(*
Nazwa:			FB_OEECycleTimes
Opis:			czasy cyklów
Wersja:			v0.1
Data:			2021-11-09
Autor:			DP
Urzadzenia:		
Konfiguracja:	
Info: 
- dodano opcje przesuwu liniowego
*)
FUNCTION_BLOCK FB_OEECycleTimes
VAR_INPUT
	bEnable: BOOL;				//Zezwolenie na pracę
	bReset:BOOL;				//Stop awaryjny nieaktywny
	tStation1CT:TIME;			//Czas cyklu stacji nr 1
	bStation1En:BOOL;			//Zezwolenie pracy stacji nr 1
	sStation1Name:STRING;		//Nazwa stacji nr 1
	tStation2CT:TIME;			//Czas cyklu stacji nr 2
	bStation2En:BOOL;			//Zezwolenie pracy stacji nr 2
	sStation2Name:STRING;		//Nazwa stacji nr 2
	tStation3CT:TIME;			//Czas cyklu stacji nr 3
	bStation3En:BOOL;			//Zezwolenie pracy stacji nr 3
	sStation3Name:STRING;		//Nazwa stacji nr 3
	tStation4CT:TIME;			//Czas cyklu stacji nr 4
	bStation4En:BOOL;			//Zezwolenie pracy stacji nr 4
	sStation4Name:STRING;		//Nazwa stacji nr 4
	tStation5CT:TIME;			//Czas cyklu stacji nr 5
	bStation5En:BOOL;			//Zezwolenie pracy stacji nr 5
	sStation5Name:STRING;		//Nazwa stacji nr 5
	tStation6CT:TIME;			//Czas cyklu stacji nr 6
	bStation6En:BOOL;			//Zezwolenie pracy stacji nr 6
	sStation6Name:STRING;		//Nazwa stacji nr 6
	tStation7CT:TIME;			//Czas cyklu stacji nr 7
	bStation7En:BOOL;			//Zezwolenie pracy stacji nr 7
	sStation7Name:STRING;		//Nazwa stacji nr 7
	tStation8CT:TIME;			//Czas cyklu stacji nr 8
	bStation8En:BOOL;			//Zezwolenie pracy stacji nr 8
	sStation8Name:STRING;		//Nazwa stacji nr 8
	tStation9CT:TIME;			//Czas cyklu stacji nr 9
	bStation9En:BOOL;			//Zezwolenie pracy stacji nr 9
	sStation9Name:STRING;		//Nazwa stacji nr 9
	tStation10CT:TIME;			//Czas cyklu stacji nr 10
	bStation10En:BOOL;			//Zezwolenie pracy stacji nr 10
	sStation10Name:STRING;		//Nazwa stacji nr 10
	tStation11CT:TIME;			//Czas cyklu stacji nr 11
	bStation11En:BOOL;			//Zezwolenie pracy stacji nr 11
	sStation11Name:STRING;		//Nazwa stacji nr 11
	tStation12CT:TIME;			//Czas cyklu stacji nr 12
	bStation12En:BOOL;			//Zezwolenie pracy stacji nr 12
	sStation12Name:STRING;		//Nazwa stacji nr 12
	tStation13CT:TIME;			//Czas cyklu stacji nr 13
	bStation13En:BOOL;			//Zezwolenie pracy stacji nr 13
	sStation13Name:STRING;		//Nazwa stacji nr 13
	tStation14CT:TIME;			//Czas cyklu stacji nr 14
	bStation14En:BOOL;			//Zezwolenie pracy stacji nr 14
	sStation14Name:STRING;		//Nazwa stacji nr 14
	tStation15CT:TIME;			//Czas cyklu stacji nr 15
	bStation15En:BOOL;			//Zezwolenie pracy stacji nr 15	
	sStation15Name:STRING;		//Nazwa stacji nr 15
	tStation16CT:TIME;			//Czas cyklu stacji nr 16
	bStation16En:BOOL;			//Zezwolenie pracy stacji nr 16	
	sStation16Name:STRING;		//Nazwa stacji nr 16
	tStation17CT:TIME;			//Czas cyklu stacji nr 17
	bStation17En:BOOL;			//Zezwolenie pracy stacji nr 17	
	sStation17Name:STRING;		//Nazwa stacji nr 17
	tStation18CT:TIME;			//Czas cyklu stacji nr 18
	bStation18En:BOOL;			//Zezwolenie pracy stacji nr 18	
	sStation18Name:STRING;		//Nazwa stacji nr 18
	tStation19CT:TIME;			//Czas cyklu stacji nr 19
	bStation19En:BOOL;			//Zezwolenie pracy stacji nr 19	
	sStation19Name:STRING;		//Nazwa stacji nr 19
	tStation20CT:TIME;			//Czas cyklu stacji nr 20
	bStation20En:BOOL;			//Zezwolenie pracy stacji nr 20	
	sStation20Name:STRING;		//Nazwa stacji nr 20
	tStation21CT:TIME;			//Czas cyklu stacji nr 21
	bStation21En:BOOL;			//Zezwolenie pracy stacji nr 21	
	sStation21Name:STRING;		//Nazwa stacji nr 21	
	tStation22CT:TIME;			//Czas cyklu stacji nr 22
	bStation22En:BOOL;			//Zezwolenie pracy stacji nr 22	
	sStation22Name:STRING;		//Nazwa stacji nr 22	
	tStation23CT:TIME;			//Czas cyklu stacji nr 23
	bStation23En:BOOL;			//Zezwolenie pracy stacji nr 23	
	sStation23Name:STRING;		//Nazwa stacji nr 23	
	tStation24CT:TIME;			//Czas cyklu stacji nr 24
	bStation24En:BOOL;			//Zezwolenie pracy stacji nr 24	
	sStation24Name:STRING;		//Nazwa stacji nr 24	
	tStation25CT:TIME;			//Czas cyklu stacji nr 25
	bStation25En:BOOL;			//Zezwolenie pracy stacji nr 25	
	sStation25Name:STRING;		//Nazwa stacji nr 25	
	tStation26CT:TIME;			//Czas cyklu stacji nr 26
	bStation26En:BOOL;			//Zezwolenie pracy stacji nr 26	
	sStation26Name:STRING;		//Nazwa stacji nr 26	
	tStation27CT:TIME;			//Czas cyklu stacji nr 27
	bStation27En:BOOL;			//Zezwolenie pracy stacji nr 27	
	sStation27Name:STRING;		//Nazwa stacji nr 27	
	tStation28CT:TIME;			//Czas cyklu stacji nr 28
	bStation28En:BOOL;			//Zezwolenie pracy stacji nr 28	
	sStation28Name:STRING;		//Nazwa stacji nr 28	
	tStation29CT:TIME;			//Czas cyklu stacji nr 29
	bStation29En:BOOL;			//Zezwolenie pracy stacji nr 29	
	sStation29Name:STRING;		//Nazwa stacji nr 29	
	tStation30CT:TIME;			//Czas cyklu stacji nr 30
	bStation30En:BOOL;			//Zezwolenie pracy stacji nr 30	
	sStation30Name:STRING;		//Nazwa stacji nr 30	
	tStation31CT:TIME;			//Czas cyklu stacji nr 31
	bStation31En:BOOL;			//Zezwolenie pracy stacji nr 31	
	sStation31Name:STRING;		//Nazwa stacji nr 31	
	
END_VAR
VAR_OUTPUT
	AsCycleTimes					:ARRAY [0..63] OF STRING;		// Tabela czasów cykli 		[symbol_stacji;czas_w_ms]
END_VAR

VAR

END_VAR

ErrorHandling();
Cycle();
ManualMovements();
Statistics();

ACTION Cycle:


//Generowanie tablicy
IF tStation1CT < T#10S THEN	AsCycleTimes[1]:=	CONCAT(sStation1Name,	CONCAT(';',DINT_TO_STRING(TIME_TO_DINT(tStation1CT))));		ELSE tStation1CT := T#10S; END_IF;

IF tStation2CT < T#10S THEN	AsCycleTimes[2]:=	CONCAT(sStation2Name,	CONCAT(';',DINT_TO_STRING(TIME_TO_DINT(tStation2CT))));		ELSE tStation1CT := T#10S; END_IF;

IF tStation3CT < T#10S THEN	AsCycleTimes[3]:=	CONCAT(sStation3Name,	CONCAT(';',DINT_TO_STRING(TIME_TO_DINT(tStation3CT))));		ELSE tStation1CT := T#10S; END_IF;

IF tStation4CT < T#10S THEN	AsCycleTimes[4]:=	CONCAT(sStation4Name,	CONCAT(';',DINT_TO_STRING(TIME_TO_DINT(tStation4CT))));		ELSE tStation4CT := T#10S; END_IF;

IF tStation5CT < T#10S THEN	AsCycleTimes[5]:=	CONCAT(sStation5Name,	CONCAT(';',DINT_TO_STRING(TIME_TO_DINT(tStation5CT))));		ELSE tStation5CT := T#10S; END_IF;

IF tStation6CT < T#10S THEN	AsCycleTimes[6]:=	CONCAT(sStation6Name,	CONCAT(';',DINT_TO_STRING(TIME_TO_DINT(tStation6CT))));		ELSE tStation6CT := T#10S; END_IF;
	
IF tStation7CT < T#10S THEN AsCycleTimes[7]:=	CONCAT(sStation7Name,	CONCAT(';',DINT_TO_STRING(TIME_TO_DINT(tStation7CT))));		ELSE tStation7CT := T#10S; END_IF;
	
IF tStation8CT < T#10S THEN AsCycleTimes[8]:=	CONCAT(sStation8Name,	CONCAT(';',DINT_TO_STRING(TIME_TO_DINT(tStation8CT))));		ELSE tStation8CT := T#10S; END_IF;
	
IF tStation9CT < T#10S THEN AsCycleTimes[9]:=	CONCAT(sStation9Name,	CONCAT(';',DINT_TO_STRING(TIME_TO_DINT(tStation9CT))));		ELSE tStation9CT := T#10S; END_IF;
	
IF tStation10CT < T#10S THEN AsCycleTimes[10]:=	CONCAT(sStation10Name,	CONCAT(';',DINT_TO_STRING(TIME_TO_DINT(tStation10CT))));	ELSE tStation10CT := T#10S; END_IF;

IF tStation11CT < T#10S THEN AsCycleTimes[11]:=	CONCAT(sStation11Name,	CONCAT(';',DINT_TO_STRING(TIME_TO_DINT(tStation11CT))));	ELSE tStation11CT := T#10S; END_IF;

IF tStation12CT < T#10S THEN AsCycleTimes[12]:=	CONCAT(sStation12Name,	CONCAT(';',DINT_TO_STRING(TIME_TO_DINT(tStation12CT))));	ELSE tStation12CT := T#10S; END_IF;

IF tStation13CT < T#10S THEN AsCycleTimes[13]:=	CONCAT(sStation13Name,	CONCAT(';',DINT_TO_STRING(TIME_TO_DINT(tStation13CT))));	ELSE tStation13CT := T#10S; END_IF;

IF tStation14CT < T#10S THEN AsCycleTimes[14]:=	CONCAT(sStation14Name,	CONCAT(';',DINT_TO_STRING(TIME_TO_DINT(tStation14CT))));	ELSE tStation14CT := T#10S; END_IF;

IF tStation15CT < T#10S THEN AsCycleTimes[15]:=	CONCAT(sStation15Name,	CONCAT(';',DINT_TO_STRING(TIME_TO_DINT(tStation15CT))));	ELSE tStation15CT := T#10S; END_IF;

IF tStation16CT < T#10S THEN AsCycleTimes[16]:=	CONCAT(sStation16Name,	CONCAT(';',DINT_TO_STRING(TIME_TO_DINT(tStation16CT))));	ELSE tStation16CT := T#10S; END_IF;

IF tStation17CT < T#10S THEN AsCycleTimes[17]:=	CONCAT(sStation17Name,	CONCAT(';',DINT_TO_STRING(TIME_TO_DINT(tStation17CT))));	ELSE tStation17CT := T#10S; END_IF;

IF tStation18CT < T#10S THEN AsCycleTimes[18]:=	CONCAT(sStation18Name,	CONCAT(';',DINT_TO_STRING(TIME_TO_DINT(tStation18CT))));	ELSE tStation18CT := T#10S; END_IF;

IF tStation19CT < T#10S THEN AsCycleTimes[19]:=	CONCAT(sStation19Name,	CONCAT(';',DINT_TO_STRING(TIME_TO_DINT(tStation19CT))));	ELSE tStation19CT := T#10S; END_IF;

IF tStation20CT < T#10S THEN AsCycleTimes[20]:=	CONCAT(sStation20Name,	CONCAT(';',DINT_TO_STRING(TIME_TO_DINT(tStation20CT))));	ELSE tStation20CT := T#10S; END_IF;

IF tStation21CT < T#10S THEN AsCycleTimes[21]:=	CONCAT(sStation21Name,	CONCAT(';',DINT_TO_STRING(TIME_TO_DINT(tStation21CT))));	ELSE tStation21CT := T#10S; END_IF;

IF tStation22CT < T#10S THEN AsCycleTimes[22]:=	CONCAT(sStation22Name,	CONCAT(';',DINT_TO_STRING(TIME_TO_DINT(tStation22CT))));	ELSE tStation22CT := T#10S; END_IF;

IF tStation23CT < T#10S THEN AsCycleTimes[23]:=	CONCAT(sStation23Name,	CONCAT(';',DINT_TO_STRING(TIME_TO_DINT(tStation23CT))));	ELSE tStation23CT := T#10S; END_IF;
	
IF tStation24CT < T#10S THEN AsCycleTimes[24]:=	CONCAT(sStation24Name,	CONCAT(';',DINT_TO_STRING(TIME_TO_DINT(tStation24CT))));	ELSE tStation24CT := T#10S; END_IF;

IF tStation25CT < T#10S THEN AsCycleTimes[25]:=	CONCAT(sStation25Name,	CONCAT(';',DINT_TO_STRING(TIME_TO_DINT(tStation25CT))));	ELSE tStation25CT := T#10S; END_IF;

IF tStation26CT < T#10S THEN AsCycleTimes[26]:=	CONCAT(sStation26Name,	CONCAT(';',DINT_TO_STRING(TIME_TO_DINT(tStation26CT))));	ELSE tStation26CT := T#10S; END_IF;

IF tStation27CT < T#10S THEN AsCycleTimes[27]:=	CONCAT(sStation27Name,	CONCAT(';',DINT_TO_STRING(TIME_TO_DINT(tStation27CT))));	ELSE tStation27CT := T#10S; END_IF;

IF tStation28CT < T#10S THEN AsCycleTimes[28]:=	CONCAT(sStation28Name,	CONCAT(';',DINT_TO_STRING(TIME_TO_DINT(tStation28CT))));	ELSE tStation28CT := T#10S; END_IF;

IF tStation29CT < T#10S THEN AsCycleTimes[29]:=	CONCAT(sStation29Name,	CONCAT(';',DINT_TO_STRING(TIME_TO_DINT(tStation29CT))));	ELSE tStation29CT := T#10S; END_IF;

IF tStation30CT < T#10S THEN AsCycleTimes[30]:=	CONCAT(sStation30Name,	CONCAT(';',DINT_TO_STRING(TIME_TO_DINT(tStation30CT))));	ELSE tStation30CT := T#10S; END_IF;

IF tStation31CT < T#10S THEN AsCycleTimes[31]:=	CONCAT(sStation31Name,	CONCAT(';',DINT_TO_STRING(TIME_TO_DINT(tStation31CT))));	ELSE tStation31CT := T#10S; END_IF;
END_ACTION

ACTION ErrorHandling:

END_ACTION

ACTION ManualMovements:

END_ACTION

ACTION Statistics:

END_ACTION

END_FUNCTION_BLOCK

(* stored: Version 1.1.0.1, ProductVersion 3.1.4026.13, FileIdentifier f45207dccd9cdddb2f244c760de4bf469eb411d1, FileSignature 4e845aef2a8a341b22efeaf01abe1ec9b05d1b3b5d8d53dc25a68e59a2dabdd8434877721504f39f1beb603aeea0e90dd4a536500e7a8a221f4e5107288d594b02e22ad73ecb9ca9decad34ff567f3a242d354c1e332166b646f690e1cbc0956ddad78356343e6bff82aad8587b8bea561623e22678181fcb62f3c1ce9bc1b3507c7428b44fc793984977013a51a863529d784bf540d412a05e37817a6b5cd2d87389ef8ef171af480398ac81d4a9016570cdc5125fe2984bb4bd041261a2376093511e86ff35fe5d691ab041d286845f78f2646c891efc18e63c24cbb46aa9d8fcf64f7b565b98218c8e861153d03b13d7649a96290c3ce3649a9ca30e00807
   POU FB_OEECycleTimes: Id {961b2418-39e3-45cc-b233-4b5a5273756c}, SpecialFunc None
   Action Cycle: Id {f6435581-9f60-43a6-8507-5e908fe1bf82}
   Action ErrorHandling: Id {8d08ea9b-3a8a-42c7-a05d-0abd149fd27a}
   Action ManualMovements: Id {8852ab39-41a6-47ba-b4a8-524830a7ab12}
   Action Statistics: Id {76c1b1be-2345-40df-b52d-74a45e42eb67} *)
